PROGRAM prgMiddle
VAR
	i: INT;
	int_LiveCount_5min:INT;								//{#lynus.ag#()}
	ton_5min: Ton;
	uint_State								AT%I* 	: UINT;		//{#lynus.ag#()}
	mtest: BOOL;

END_VAR

i:= i+1;
ton_5min( 	In := NOT ton_5min.Q,
			PT := T#5M);
IF ton_5min.Q THEN
	int_LiveCount_5min := int_LiveCount_5min+1;
END_IF

prgHeatPump();
prgRoomVentilaton();

END_PROGRAM

(* stored: Version 1.1.0.1, ProductVersion 3.1.4024.12
   POU prgMiddle: Id {1ae37f63-3cea-4a0e-998c-c679029efd1a}, SpecialFunc None *)
